Staubli VAL3: clkDoModules.pgx

program clkDoModules()
begin
  bDoModules = true
end
